PROGRAM P_Demo_PSTRING_TO_STRING
VAR
    sRealValue           : STRING(80) := 'Hello PLC'; // 模拟 wire 缓冲区中的 STRING 字段
    pSTRINGField         : POINTER TO STRING(80); // 业务侧先算好的字段地址（ADR 或 pBase+nOff）
    bExtractField        : BOOL; // 在线置 TRUE 触发一次解析
    sRealValue_extracted : STRING(80); // 解析后的副本，供业务逻辑使用
END_VAR

// ============================================================
// Tc2_Utilities.PSTRING_TO_STRING 演示程序（FUNCTION）
// ============================================================
// 场景：从一段二进制 wire 缓冲区里按偏移取 STRING 字段（Modbus/CAN/ADS Raw）。
// 价值：替代手写 pField + nOff + ^ 指针算术；一次调用取值，少打错符号。
// 验证：在线写 sRealValue := 'Hello PLC'；bExtractField := TRUE；
//       下一周期 sRealValue_extracted 应等于 sRealValue。
// ============================================================

// 业务代码通常已经算好字段地址（pBase + 协议偏移）；演示用 ADR 等价
pSTRINGField := ADR(sRealValue);

IF bExtractField AND pSTRINGField <> 0 THEN
    // 单次完整调用：避免手写 ^ 解引用，统一风格便于和字节序转换串联
    sRealValue_extracted := PSTRING_TO_STRING(pSTRINGField);
    bExtractField := FALSE;
END_IF;

END_PROGRAM

(* stored: Version 1.1.0.1, ProductVersion 3.1.4024.5
   POU P_Demo_PSTRING_TO_STRING: Id {56ea05b4-5b22-5b9e-9d57-cfb72587143a}, SpecialFunc None *)
